// TIA Portal V17 export
// export: Created 2024-08-09T12:53:13.3895526Z, ExportSetting WithDefaults, DisplayName Totally Integrated Automation Portal, DisplayVersion V17 Update 7, DisplayName TIA Portal Openness, DisplayVersion V17 Update 7, DisplayName TIA Portal Version Control Interface, DisplayVersion V17, DisplayName STEP 7 Professional, DisplayVersion V17 Update 7, DisplayName STEP 7 Safety, DisplayVersion V17 Update 6, DisplayName WinCC Professional, DisplayVersion V17 Update 7
VAR_GLOBAL   // PLC tag table "BROYAGE"
END_VAR
VAR_GLOBAL CONSTANT   // user constants
   NIV_BR_DEBUT_LOT : USInt := 1;
   NIV_BR_COND_ATTEINTES : USInt := 3;
   NIV_BR_PRET : USInt := 5;
   NIV_BR_VIT_ATTEINTE : USInt := 10;
   NIV_BR_ALIM_MARCHE : USInt := 20;
   NIV_BR_FIN_PRD_BR : USInt := 30;
   NIV_BR_ARR_ALIM : USInt := 40;
   NIV_BR_FIN_PM_SOUS_BR : USInt := 50;
   NIV_BR_FIN_LOT : USInt := 255;
END_VAR
